TYPE ST_InstruOnChipData :
STRUCT

	// ID
	m_InstruID: INT:=0;
	
	// series number
	m_InstruseriesNum : ULINT:=0;
	
	// current and max usage counts
	m_InstruUsageCounts :ULINT;
	m_InstrumaxUsageCounts :ULINT:=20;
	
	//Instrument Zero augular offset
	m_InstruPos:Vec5d;
	
	//Instrument state
	m_InstruReadSucceed:BOOL;
	
	//Instrument Clamp Error
	m_Error:BOOL;
	m_ErrorID:INT;//1器械类型错误、2器械使用次数超限、3两个内窥镜
	
	m_InstruPurpose :ULINT;
	m_InstruPurposeTime :ULINT;
END_STRUCT
END_TYPE

(* stored: Version 1.1.0.1, ProductVersion 3.1.4024.11
   DUT ST_InstruOnChipData: Id {24a5a89b-c2a6-4796-bae1-11e8082d9094} *)
